{attribute 'qualified_only'}
{attribute 'strict'}
{attribute 'to_string'}

TYPE e400VSupplySource :
(
	none := 0,
	grid := 1,
	CEE := 2
);
END_TYPE

(* stored: Version 1.1.0.1, ProductVersion 3.1.4026.18
   DUT e400VSupplySource: Id {5d549a7f-cf6f-4e1e-b3e4-693958cdab6d} *)
